ABB RobotStudio station: standard test station.rsstn

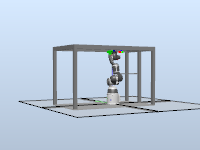
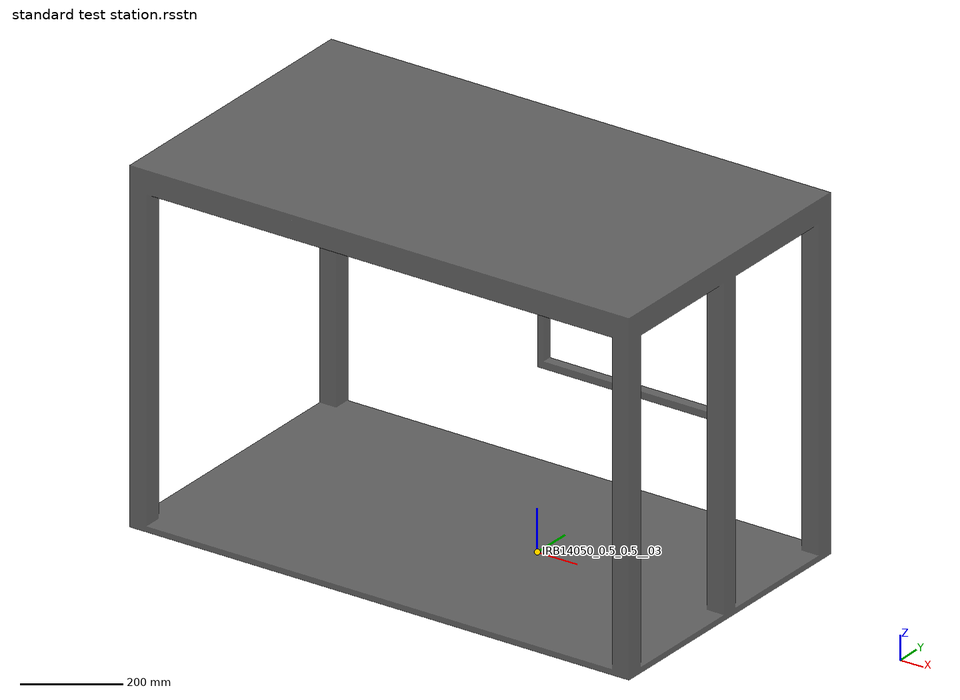
[picture v1: parts stored in the station drawn from their meshes, with robot base, taught points and paths (robot models come from the ABB library and are not in the file)]
Station standard test station (saved by RobotStudio 21.2.9526.0)
Controller Controller2
  mechanical unit ROB_1: IRB14050_0.5_0.5__03, 6 joints, base frame (0, 0, 0) mm
  mechanical unit ROB_1_7: IRB14050_0.5_0.5__03, 1 joints, base frame (0, 0, 0) mm
Layout (positions relative to the parent item):
  - IRB14050_0.5_0.5__03 [mechanism, from Robots\IRB14050_0.5_0.5__03.rslib] at (0, 0, 0) mm; joint values [1.2249, -1.6563, 0.1074, 0.2081, -0.1684, 1.4684, -0.6594] (rad or m)
  - SAY_tool_old_licens [mechanism, from Robot Studio\SAY_tool_old_licens.rslib] at (-102.05, -209.66, 645) mm, rotated rx -90 ry 45 rz -30 deg
  - roof [part], size 1180 x 680 x 12 mm
  - horizontal_pole_1 [part], size 1180 x 40 x 40 mm
  - horizontal_pole_2 [part], size 1180 x 40 x 40 mm
  - horizontal_pole_3 [part], size 40 x 600 x 40 mm
  - horizontal_pole_4 [part], size 40 x 600 x 40 mm
  - cylinder [part], size 120 x 119.8 x 120 mm
  - vertical_pole_1 [part], size 40 x 40 x 743 mm
  - vertical_pole_2 [part], size 40 x 40 x 743 mm
  - middle_vertical_pole [part], size 40 x 40 x 743 mm
  - vertical_pole_3 [part], size 40 x 40 x 743 mm
  - vertical_pole_4 [part], size 40 x 40 x 743 mm
  - sender_pole [part], size 430 x 22.5 x 15 mm
  - linear_actuator [part], size 15 x 22.5 x 208 mm
  - floor [part], size 1180 x 680 x 12 mm
  - Frame_antenna [frame] at (-20.86, -20.86, 110) mm, rotated rx 0 ry 0 rz 45 deg
  - Frame_laser [frame] at (-46.99, -23.72, 82.6) mm, rotated rx 0 ry 0 rz 45 deg
  - Frame_calibration [frame] at (-41.72, -43.13, 58.23) mm, rotated rx 0 ry -90 rz 45 deg
Attachment: SAY_tool_old_licens is attached to IRB14050_0.5_0.5__03 / Link7
Collision set robot_cylinder: IRB14050_0.5_0.5__03 against cylinder, near miss 0 m
Collision set robot_linear_act: IRB14050_0.5_0.5__03 against linear_actuator, near miss 0 m
Collision set robot_horizontal_1: IRB14050_0.5_0.5__03 against horizontal_pole_1, near miss 0 m
Collision set robot_horizontal_2: IRB14050_0.5_0.5__03 against horizontal_pole_2, near miss 0 m
Collision set robot_middle_pole: IRB14050_0.5_0.5__03 against middle_vertical_pole, near miss 0 m
Collision set robot_roof: IRB14050_0.5_0.5__03 against roof, near miss 0 m
Collision set robot_sender_pole: IRB14050_0.5_0.5__03 against sender_pole, near miss 0 m
Collision set robot_horizontal_3: IRB14050_0.5_0.5__03 against horizontal_pole_3, near miss 0 m
Collision set robot_horizontal_4: IRB14050_0.5_0.5__03 against horizontal_pole_4, near miss 0 m
Collision set robot_vertical_1: IRB14050_0.5_0.5__03 against vertical_pole_1, near miss 0 m
Collision set robot_vertical_2: IRB14050_0.5_0.5__03 against vertical_pole_2, near miss 0 m
Collision set robot_vertical_3: IRB14050_0.5_0.5__03 against vertical_pole_3, near miss 0 m
Collision set robot_vertical_4: IRB14050_0.5_0.5__03 against vertical_pole_4, near miss 0 m
Collision set tool_cylinder: SAY_tool_old_licens against cylinder, near miss 0 m
Collision set tool_floor: SAY_tool_old_licens against floor, near miss 0 m
Collision set tool_horizontal_1: SAY_tool_old_licens against horizontal_pole_1, near miss 0 m
Collision set tool_horizontal_2: SAY_tool_old_licens against horizontal_pole_2, near miss 0 m
Collision set tool_horizontal_3: SAY_tool_old_licens against horizontal_pole_3, near miss 0 m
Collision set tool_horizontal_4: SAY_tool_old_licens against horizontal_pole_4, near miss 0 m
Collision set tool_linear-act: SAY_tool_old_licens against linear_actuator, near miss 0 m
Collision set tool_middle_vertical: SAY_tool_old_licens against middle_vertical_pole, near miss 0 m
Collision set tool_roof: SAY_tool_old_licens against roof, near miss 0 m
Collision set tool_sender: SAY_tool_old_licens against sender_pole, near miss 0 m
Collision set tool_vertical_1: SAY_tool_old_licens against vertical_pole_1, near miss 0 m
Collision set tool_vertical_2: SAY_tool_old_licens against vertical_pole_2, near miss 0 m
Collision set tool_vertical_3: SAY_tool_old_licens against vertical_pole_3, near miss 0 m
Collision set tool_vertical_4: SAY_tool_old_licens against vertical_pole_4, near miss 0 m
Targets, tools, work objects and paths stored in the station, written as RAPID:
! task T_ROB1
MODULE SERVER
  PERS tooldata antenna_tcp:=[TRUE,[[-20.86,-20.859,110],[0.923879533,0,0,0.382683432]],[0.1,[-18.786,-18.883,43.148],[1,0,0,0],0,0,0]];
  PERS tooldata laser_tcp:=[TRUE,[[-46.987,-23.723,82.6],[0.923879533,0,0,0.382683432]],[0.1,[-18.786,-18.883,43.148],[1,0,0,0],0,0,0]];
  PERS tooldata calibration_tcp:=[TRUE,[[-41.72,-43.133,58.227],[0.653281482,0.27059805,-0.653281482,0.27059805]],[0.1,[-18.786,-18.883,43.148],[1,0,0,0],0,0,0]];
ENDMODULE

! task T_ROB1
MODULE Module1
  CONST robtarget Target_10:=[[149.372616104,17.449358706,706.001461714],[0.000006556,0.000007919,0.000012199,-1],[-1,-1,0,4],[0.000004243,9E+09,9E+09,9E+09,9E+09,9E+09]];
ENDMODULE

